(*******************************************************************************
                          protoc-gen-twincat V0.0.0.0                           
                  https://github.com/TcHaxx/protoc-gen-twincat                  
*******************************************************************************)
{attribute 'qualified_only'}
{attribute 'strict'}
{attribute 'to_string'}
// Enum with enum_prefix and enum_integer_type options
TYPE E_Color :
(
	COLOR_DEFAULT := 0,
	COLOR_RED := 1,
	COLOR_GREEN := 2,
	COLOR_BLUE := 3
) WORD;
END_TYPE

(* stored: Version 1.1.0.1
   DUT E_Color: Id 418a1aef-fe0f-4ca2-8f79-287eb3353c4e *)
